{attribute 'enable_dynamic_creation'}
FUNCTION_BLOCK Rectangle EXTENDS Disposable IMPLEMENTS I_DrawableShape
VAR
	_width: INT;
    _height: INT;
END_VAR

METHOD Clone : I_DrawableShape
VAR
	pRectangle : POINTER TO Rectangle;
END_VAR
pRectangle := __NEW(Rectangle);
pRectangle^.Width := Width;
pRectangle^.Height := Height;
Clone := pRectangle^;
END_METHOD

METHOD Draw
VAR
	str_width : STRING;
	str_height : STRING;
	str : STRING;
END_VAR
str_width := CONCAT(STR1 := 'width: ', STR2 := TO_STRING(Width));
str_height := CONCAT(STR1 := 'height: ', STR2 := TO_STRING(Height));
str := CONCAT(STR1 := str_width, STR2 := str_height);
ADSLOGSTR(msgCtrlMask := ADSLOG_MSGTYPE_HINT, msgFmtStr := 'Draw Rectangle with:  %s', strArg := str);
END_METHOD

PROPERTY PUBLIC Height : INT
GET
Height := _height;
END_GET
SET // PUBLIC
_height := Height;
END_SET
END_PROPERTY

PROPERTY PUBLIC Width : INT
GET
Width := _width;
END_GET
SET // PUBLIC
_width := Width;
END_SET
END_PROPERTY

END_FUNCTION_BLOCK

(* stored: Version 1.1.0.1, ProductVersion 3.1.4024.12
   POU Rectangle: Id {5fab8419-38ec-4aa0-8ae7-fe6ce34dda2e}, SpecialFunc None
   Method Clone: Id {d393242f-6ae7-4dca-af0b-60b70a6eaa0e}
   Method Draw: Id {d8fa6ad4-ea28-4c15-ab4b-56aa068bd55b}
   Property Height: Id {ab99e11c-9a78-4285-bdf1-cf57d8eff6b0}
   Get Get: Id {0d5a2626-dceb-4d2b-9482-c397d81644a4}
   Set Set: Id {2730e795-16db-4b57-b07b-803afb9c281d}
   Property Width: Id {d396d12a-4ac7-4a07-8804-d7ad3f55cf54}
   Get Get: Id {40509c85-7ea1-475d-837f-e80992516ae4}
   Set Set: Id {401e5243-7204-466b-9a08-420f881b0269} *)
